TEXTLIST CRAH_Isolator_Status
  0 = 'OFF'
  1 = 'ON'
   = ''
END_TEXTLIST

(* stored: Version 1.1.0.1, ProductVersion 3.1.4024.12
   TextList CRAH_Isolator_Status: Id {7c5e8e8a-0bbf-4792-b4ef-91cbcc32f60c} *)
